TYPE Variablen :
STRUCT
	q1		: ARRAY[0..7] OF BYTE;
	q2		: ARRAY[0..7] OF BYTE;
	q3		: ARRAY[0..7] OF BYTE;
	q4		: ARRAY[0..7] OF BYTE;
	q5		: ARRAY[0..7] OF BYTE;
	q6		: ARRAY[0..7] OF Byte;
END_STRUCT
END_TYPE

(* stored: Version 1.1.0.1
   DUT Variablen: Id {d516b813-01d3-4de4-b44b-127cf89f0b33} *)
